Omron CX-Programmer project NewProject (CX-Programmer 9.61)

# PLC COUNTER: CP1L M
; TES COUNTER

## Global symbols (name address type ; comment)
0.00 BOOL  ; START
0.01 BOOL  ; RESET
100.00 BOOL  ; LAMPU
C0000 BOOL  ; COUNT #4

## Program NewProgram1 (cyclic task 0)

### Section Section1

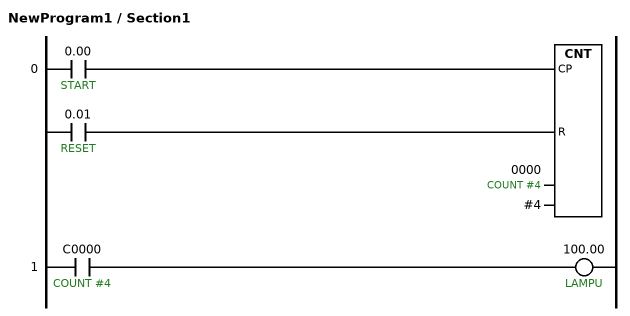
; rung 0
LD 0.00  ; START
LD 0.01  ; RESET
CNT 0000 #4  ; COUNT #4
; rung 1
LD C0000  ; COUNT #4
OUT 100.00  ; LAMPU

### Section END
; rung 0
END(001)